(* CODESYS project MC508.project
   Title: MC508
   CompiledLibraryCompatibilityVersion: LeadSysStudio V3.5 SP15 Patch 4

Project tree, tasks and I/O mapping:
  Device : MC508, Leadshine Technology Co., Ltd., order no. 508101, version 3.5.15.40
      settings: RetainMode = 0; RetainStartAddr = 20480; RetainEndAddr = 524288; RetainSize = 524288
    application Application
      libraries: Standard, * (System); VisuDialogs, * (System); LS_ModbusMasterlib, 0.0.0.2 (Leadshine Technology Co.Ltd)
      task MainTask (cyclic, interval 500 µs, priority 1) calls main
      program main [ST]: io, vfd_setup, motion, save_apply, vfd, save_check, cut, supply, extract, work, stick
      visualisation Visualization
      Symbols
      function StateNext [ST]
      Object/
        data type Cylinder
        data type Button
      Enum/
        data type State
        data type VFDType
      DataMain/
        data type HMIData
        data type SaveData
        data type VFDData
      DataWork/
        data type CutData
        data type SupplyData
        data type ExtractData
        data type WorkData
        data type StickData
    Device Diagnose
    Network Configuration
      LocalBus Config
    Resource Usage
    SoftMotion General Axis Pool
      LS_Axis_0 : Axis, 3S - Smart Software Solutions GmbH, order no. 1805, version 4.0.0.0
          settings: eRampType = 3; fSWLimitPositive = 0.0
      LS_Axis_1 : Axis, 3S - Smart Software Solutions GmbH, order no. 1805, version 4.0.0.0
          settings: wDriveID = 2; eRampType = 3
    High_Speed_IO_Module : High Speed IO, Leadshine Technology Co., Ltd., version 3.5.15.40
        settings: HS_IO_Mode_0.High Out IO Mode 0 = 65537; HS_IO_Mode_0.High Out IO Mode 1 = 65537; Axis_Mask = 3; Ioout_Mask = 15; Axis_0_Pulse_FPGA_Config.Axis Ratio Nume = 1000; Axis_0_Pulse_FPGA_Config.Axis Ratio Denom = 1000; Axis_1_Pulse_FPGA_Config.Axis Ratio Nume = 1000; Axis_1_Pulse_FPGA_Config.Axis Ratio Denom = 50000
        unmapped channels: Genral_IO_IN, Genral_IO_Out
    LocalBus_Master_Module : LocalBus Master, Leadshine Technology Co., Ltd., version 3.5.15.40
  text list GlobalTextList
*)

// Device/Application/DataMain/HMIData
TYPE HMIData :
STRUCT
	plc_ready: BOOL;
	hmi_ready: BOOL;
	run: BOOL;
	stop: BOOL;
	//
	supply_run_press: BOOL;
	supply_run_glue: BOOL;
	supply_run_conveyer: BOOL;
	supply_run_roll: BOOL;
	stick_run_press: BOOL;
	stick_run_roll: BOOL;
	cut_run: BOOL;
	extract_run: BOOL;
	//
	supply_press_a: BOOL;
	supply_press_b: BOOL;
	stick_press: BOOL;
	cut_press: BOOL;
	//
	vfds_run: ARRAY[0..15] OF BOOL;
	//
	save_data: SaveData;
	save: BOOL;
	save_need_check: BOOL;
	save_need: BOOL;
	//
	view_stop: BOOL;
	view_halt: BOOL;
	view_can_run: BOOL;
	view_can_stop: BOOL;
	view_supply_roll_is_long: BOOL;
	view_supply_roll_is_short: BOOL;
	view_supply_select_roll: BOOL;
	view_stick_foil_in: BOOL;
	view_stick_roll_speed_micron_per_sec: UDINT;
	view_cut_foil_in: BOOL;
	view_cut_position: DINT;
	view_cut_speed_micron_per_sec: UDINT;
	view_cut_servo_is_ready: BOOL;
	view_cut_servo_is_home: BOOL;
	view_extract_foil_in: BOOL;
	view_extract_reach: BOOL;
	//
	view_state_main: INT;
	view_state_work: INT;
	//
	view_state_supply_press: INT;
	view_state_supply_glue: INT;
	view_state_supply_conveyer: INT;
	view_state_supply_roll: INT;
	view_state_stick_press: INT;
	view_state_stick_roll: INT;
	view_state_cut: INT;
	view_state_extract: INT;
	//
	view_vfds_f_target: ARRAY[0..15] OF UINT;
END_STRUCT
END_TYPE

// Device/Application/Enum/State
{attribute 'qualified_only'}
{attribute 'strict'}
TYPE State : (
	NONE := 0,
	RST := 1,
	RST_DONE := 50,
	HOME := 51,
	HOME_FORWARD := 71,
	HOME_DONE := 99,
	READY := 100,
	RUN := 101,
	RUN_ING := 200
);
END_TYPE

// Device/Application/DataMain/SaveData
TYPE SaveData :
STRUCT
	set_done: BOOL;
	main_frequency: UINT;
	stick_speed_factor: UDINT;
	stick_roll_gear_ratio: UDINT;
	stick_roll_diameter_micron: UDINT;
	stick_stop_distance_micron: UDINT; // distance after panel's tail move out of sensor
	cut_angle_radian: UDINT;
	cut_length_micron: UDINT;
	cut_accel_decel_time: UINT;
	cut_run_distance_micron: UINT; // distance after panel's head enter sensor
	vfds_frequency_factor: ARRAY[0..15] OF UINT;
END_STRUCT
END_TYPE

// Device/Application/DataWork/CutData
TYPE CutData :
STRUCT
	state: INT;
	press: Cylinder;
	servo_on: BOOL;
	servo_is_ready: BOOL;
	servo_is_home: BOOL;
	foil_in_rise: R_TRIG;
	foil_in_fall: F_TRIG;
	blade_vfd_id: USINT;
	speed_target: LREAL; // micron per sec
	speed_factor: LREAL; // speed_factor = current_velocity / target_velocity
	speed_factor_active: BOOL;
	travel_length_micron: LREAL; // travel_length = cut_length / cos(angle_radian)
	accel_decel_time: LREAL;
	angle_radian: LREAL;
	run: Button;
	//
	sin_cut_angle: LREAL;
	home_zero_position: LREAL;
	stick_axis_target_position: LREAL;
END_STRUCT
END_TYPE

// Device/Application/DataMain/VFDData
TYPE VFDData :
STRUCT
	vfds_type: ARRAY[0..15] OF INT;
	i: USINT;
	i_control: UINT;
	i_frequency: DINT;
END_STRUCT
END_TYPE

// Device/Application/DataWork/SupplyData
TYPE SupplyData :
STRUCT
	state_press: INT;
	press_a: Cylinder;
	press_b: Cylinder;
	run_press: Button;
	//
	state_glue: INT;
	glues_vfd_id: ARRAY[0..1] OF USINT;
	run_glue: Button;
	//
	state_conveyer: INT;
	conveyers_vfd_id: ARRAY[0..1] OF USINT;
	run_conveyer: Button;
	//
	state_roll: INT;
	rolls_vfd_id: ARRAY[0..1] OF USINT;
	roll_index: USINT;
	roll_is_long: BOOL;
	roll_is_short: BOOL;
	roll_is_short_timer: TON;
	select_roll: BOOL;
	run_roll: Button;
END_STRUCT
END_TYPE

// Device/Application/DataWork/ExtractData
TYPE ExtractData :
STRUCT
	state: INT;
	foil_in_rise: R_TRIG;
	reach_rise: R_TRIG;
	conveyers_vfd_id: ARRAY[0..1] OF USINT;
	blades_vfd_id: ARRAY[0..1] OF USINT;
	run: Button;
END_STRUCT
END_TYPE

// Device/Application/DataWork/WorkData
TYPE WorkData :
STRUCT
	state: INT;
	run: Button;
	can_run: BOOL;
	stop: Button;
	can_stop: BOOL;
	halt: Button;
END_STRUCT
END_TYPE

// Device/Application/DataWork/StickData
TYPE StickData :
STRUCT
	state_press: INT;
	state_roll: INT;
	press: Cylinder;
	foil_in_rise: R_TRIG;
	foil_in_fall: F_TRIG;
	run_press: Button;
	run_roll: Button;
	speed_target: LREAL; // 1000 ppr -> 3000 rpm = 50_000
	speed_micron_per_sec: LREAL;
	//
	micron_per_servo_round: LREAL;
	stop_distance: LREAL;
END_STRUCT
END_TYPE

// Device/Application/Object/Cylinder
TYPE Cylinder :
STRUCT
	on: BOOL;
	n_timer: TON;
	p_timer: TON;
END_STRUCT
END_TYPE

// Device/Application/Object/Button
TYPE Button :
STRUCT
	rise: R_TRIG;
	fall: F_TRIG;
END_STRUCT
END_TYPE

// Device/Application/Enum/VFDType
{attribute 'qualified_only'}
{attribute 'strict'}
TYPE VFDType :
(
	NORMAL := 0,
	SPINDLE := 1,
	CUSTOM := 2
);
END_TYPE

// Device/Application/main
PROGRAM main
VAR
	axis_stick: POINTER TO SM3_Basic.AXIS_REF_VIRTUAL_SM3;
	axis_stick_power: MC_Power;
	axis_stick_stop: MC_Stop;
	axis_stick_reset: MC_Reset;
	axis_stick_set_position: MC_SetPosition;
	axis_stick_mv: MC_MoveVelocity;
	axis_stick_fv: SMC_FollowVelocity;
	//
	axis_cut: POINTER TO SM3_Basic.AXIS_REF_VIRTUAL_SM3;
	axis_cut_power: MC_Power;
	axis_cut_stop: MC_Stop;
	axis_cut_reset: MC_Reset;
	axis_cut_set_position: MC_SetPosition;
	axis_cut_mabs: MC_MoveAbsolute;
	//
	state_main: INT;
	main_save: Button;
	supply_data: SupplyData;
	stick_data: StickData;
	cut_data: CutData;
	extract_data: ExtractData;
	work_data: WorkData;
	hmi_data: HMIData;
	//
	vfd_master: LS_ModbusMaster;
	vfd_para: SerialCommunicationPara;
	vfd_configs: ARRAY [0..127] OF ModbusConfig;
	vfd_data: VFDData;
END_VAR

VAR CONSTANT
	c_vfd_count: BYTE := 11;
	c_main_frequency_min: UINT := 10_00;
	c_main_frequency_max: UINT := 50_00;
	c_axis_stick_max_speed: LREAL := 3000.0 * 1000.0 / 60.0; // 3000rpm, 1000 ppr at servo
	c_axis_cut_max_speed: LREAL := 4920.0 * 50_000.0 / 60.0; // 4920rpm, 1000 ppr at servo
	c_axis_cut_home_speed_micron_per_sec: LREAL := 20_000.0;
	c_axis_cut_home_offset_micron: LREAL := 10_000.0;
	c_axis_stick_ramp_time_sec: LREAL := 0.1;
	c_dt: LREAL := 0.000_500;
END_VAR

VAR RETAIN
	save_data: SaveData;
END_VAR

CASE state_main OF
	State.NONE:
		axis_stick := ADR(LS_Axis_0);
		axis_cut := ADR(LS_Axis_1);
		supply_data.press_a.on := TRUE;
		axis_stick_fv.fSetVelocity := 0.0;
		vfd_setup();
		StateNext(state_main);
	1:
		axis_stick_power.Enable := TRUE;
		axis_stick_power.bDriveStart := TRUE;
		axis_stick_power.bRegulatorOn := TRUE;
		axis_cut_power.Enable := TRUE;
		axis_cut_power.bDriveStart := TRUE;
		axis_cut_power.bRegulatorOn := TRUE;
		StateNext(state_main);
	2:
		IF NOT save_data.set_done THEN
			save_data.set_done := TRUE;
			save_data.main_frequency := 50_00;
			save_data.stick_speed_factor := 1_000;
			save_data.stick_roll_gear_ratio := 20_000;
			save_data.stick_roll_diameter_micron := 120_000;
			save_data.stick_stop_distance_micron := 0_001;
			save_data.cut_angle_radian := 0_230_500;
			save_data.cut_length_micron := 290_000;
			save_data.cut_accel_decel_time := 0_100;
			save_data.cut_run_distance_micron := 20_000;
			//
			save_data.vfds_frequency_factor[supply_data.glues_vfd_id[0]] := 1_000;
			save_data.vfds_frequency_factor[supply_data.glues_vfd_id[1]] := 1_000;
			save_data.vfds_frequency_factor[supply_data.conveyers_vfd_id[0]] := 1_000;
			save_data.vfds_frequency_factor[supply_data.conveyers_vfd_id[1]] := 1_000;
			save_data.vfds_frequency_factor[supply_data.rolls_vfd_id[0]] := 0_500;
			save_data.vfds_frequency_factor[supply_data.rolls_vfd_id[1]] := 0_500;
			save_data.vfds_frequency_factor[cut_data.blade_vfd_id] := 50_00;
			save_data.vfds_frequency_factor[extract_data.conveyers_vfd_id[0]] := 50_00;
			save_data.vfds_frequency_factor[extract_data.conveyers_vfd_id[1]] := 50_00;
			save_data.vfds_frequency_factor[extract_data.blades_vfd_id[0]] := 200_00;
			save_data.vfds_frequency_factor[extract_data.blades_vfd_id[1]] := 200_00;
		END_IF
		StateNext(state_main);
	3:
		save_apply();
		StateNext(state_main);
	4:
		hmi_data.plc_ready := TRUE;
		work_data.state := State.RST;
		state_main := State.RUN_ING;
	State.RUN_ING:
		motion();
		io();
		vfd();
		work();
		supply();
		stick();
		cut();
		extract();
END_CASE

ACTION io:
work_data.can_run := work_data.stop.fall.CLK AND work_data.halt.rise.CLK AND work_data.state = State.READY;
work_data.can_stop := work_data.state >= State.RUN;
////////////
//HMI DOWN//
///////////
IF hmi_data.hmi_ready THEN
	////////
	//WORK//
	////////
	work_data.run.rise(CLK:= hmi_data.run, Q=> );
	IF work_data.run.rise.Q AND work_data.can_run THEN
		work_data.state := State.RUN;
	END_IF
	work_data.stop.rise(CLK:= hmi_data.stop, Q=> );
	IF work_data.stop.rise.Q AND work_data.can_stop THEN
		work_data.state := State.RST;
	END_IF
	//////////
	//SUPPLY//
	//////////
	supply_data.run_press.rise(CLK:= hmi_data.supply_run_press, Q=> );
	IF supply_data.run_press.rise.Q THEN
		CASE supply_data.state_press OF
			State.NONE:
				supply_data.state_press := State.RST;
			State.READY:
				supply_data.state_press := State.RUN;
			State.RUN_ING:
				supply_data.state_press := State.RST;
		END_CASE
	END_IF
	supply_data.run_glue.rise(CLK:= hmi_data.supply_run_glue, Q=> );
	IF supply_data.run_glue.rise.Q THEN
		CASE supply_data.state_glue OF
			State.NONE:
				supply_data.state_glue := State.RST;
			State.READY:
				supply_data.state_glue := State.RUN;
			State.RUN_ING:
				supply_data.state_glue := State.RST;
		END_CASE
	END_IF
	supply_data.run_conveyer.rise(CLK:= hmi_data.supply_run_conveyer, Q=> );
	IF supply_data.run_conveyer.rise.Q THEN
		CASE supply_data.state_conveyer OF
			State.NONE:
				supply_data.state_conveyer := State.RST;
			State.READY:
				supply_data.state_conveyer := State.RUN;
			State.RUN_ING:
				supply_data.state_conveyer := State.RST;
		END_CASE
	END_IF
	supply_data.run_roll.rise(CLK:= hmi_data.supply_run_roll, Q=> );
	IF supply_data.run_roll.rise.Q THEN
		CASE supply_data.state_roll OF
			State.NONE:
				supply_data.state_roll := State.RST;
			State.READY:
				supply_data.state_roll := State.RUN;
			State.RUN_ING:
				supply_data.state_roll := State.RST;
		END_CASE
	END_IF
	/////////
	//STICK//
	/////////
	stick_data.run_press.rise(CLK:= hmi_data.stick_run_press, Q=> );
	IF stick_data.run_press.rise.Q THEN
		CASE stick_data.state_press OF
			State.NONE:
				stick_data.state_press := State.RST;
			State.READY:
				stick_data.state_press := State.RUN;
			State.RUN_ING:
				stick_data.state_press := State.RST;
		END_CASE
	END_IF
	stick_data.run_roll.rise(CLK:= hmi_data.stick_run_roll, Q=> );
	IF stick_data.run_roll.rise.Q THEN
		CASE stick_data.state_roll OF
			State.NONE:
				stick_data.state_roll := State.RST;
			State.RST_DONE:
				stick_data.state_roll := State.HOME;
			State.HOME_DONE:
				stick_data.state_roll := State.READY;
			State.READY:
				stick_data.state_roll := State.RST;
		END_CASE
	END_IF
	///////
	//CUT//
	///////
	cut_data.run.rise(CLK:= hmi_data.cut_run, Q=> );
	IF cut_data.run.rise.Q THEN
		CASE cut_data.state OF
			State.NONE:
				cut_data.state := State.RST;
			State.RST_DONE:
				cut_data.state := State.HOME;
			State.HOME_DONE:
				cut_data.state := State.READY;
			State.READY:
				cut_data.state := State.RST;
		END_CASE
	END_IF
	///////////
	//EXTRACT//
	///////////
	extract_data.run.rise(CLK:= hmi_data.extract_run, Q=> );
	IF extract_data.run.rise.Q THEN
		CASE extract_data.state OF
			State.NONE:
				extract_data.state := State.RST;
			State.RST_DONE:
				extract_data.state := State.HOME;
			State.HOME_DONE:
				extract_data.state := State.READY;
			State.READY:
				extract_data.state := State.RST;
		END_CASE
	END_IF
	////////
	//SAVE//
	////////
	IF hmi_data.save_need_check THEN
		save_check();
		hmi_data.save_need_check := FALSE;
	END_IF
	main_save.rise(CLK:= hmi_data.save, Q=> );
	IF main_save.rise.Q THEN
		save_data := hmi_data.save_data;
		save_apply();
		hmi_data.save_need := FALSE;
		hmi_data.save := FALSE;
	END_IF
END_IF
/////////
//INPUT//
/////////
supply_data.roll_is_long := %IX0.4;
supply_data.roll_is_short := %IX0.5;
work_data.halt.rise(CLK:= %IX1.4, Q=> );
supply_data.select_roll := %IX1.5;
//
stick_data.foil_in_rise(CLK:= NOT %IX0.6, Q=> );
stick_data.foil_in_fall(CLK:= stick_data.foil_in_rise.CLK, Q=> );
//
cut_data.servo_is_ready := %IX0.1;
cut_data.servo_is_home := NOT %IX0.7;
cut_data.foil_in_rise(CLK:= %IX1.0, Q=> );
cut_data.foil_in_fall(CLK:= cut_data.foil_in_rise.CLK, Q=> );
//
extract_data.foil_in_rise(CLK:= %IX1.1, Q=> );
extract_data.reach_rise(CLK:= %IX1.2, Q=> );
//
work_data.stop.fall(CLK:= %IX1.7, Q=> );
IF work_data.stop.fall.Q AND work_data.can_stop THEN
	work_data.state := State.RST;
END_IF
//
supply_data.press_a.n_timer(IN:= NOT supply_data.press_a.on, PT:= , Q=> , ET=> );
supply_data.press_a.p_timer(IN:= supply_data.press_a.on, PT:= , Q=> , ET=> );
supply_data.press_b.n_timer(IN:= NOT supply_data.press_b.on, PT:= , Q=> , ET=> );
supply_data.press_b.p_timer(IN:= supply_data.press_b.on, PT:= , Q=> , ET=> );
supply_data.roll_is_short_timer(IN:= supply_data.roll_is_short, PT:= , Q=> , ET=> );
stick_data.press.n_timer(IN:= NOT stick_data.press.on, PT:= , Q=> , ET=> );
stick_data.press.p_timer(IN:= stick_data.press.on, PT:= , Q=> , ET=> );
cut_data.press.n_timer(IN:= NOT cut_data.press.on, PT:= , Q=> , ET=> );
cut_data.press.p_timer(IN:= cut_data.press.on, PT:= , Q=> , ET=> );
//////////
//OUTPUT//
//////////
%QX1.4 := NOT supply_data.press_a.on;
%QX1.5 := supply_data.press_b.on;
%QX1.6 := stick_data.press.on;
%QX1.2 := cut_data.servo_on;
%QX1.7 := NOT cut_data.press.on;
//////////
//HMI UP//
//////////
IF hmi_data.hmi_ready THEN
	hmi_data.view_stop := work_data.stop.fall.CLK;
	hmi_data.view_halt := work_data.halt.rise.CLK;
	hmi_data.view_can_run := work_data.can_run;
	hmi_data.view_can_stop := work_data.can_stop;
	hmi_data.view_supply_roll_is_long := supply_data.roll_is_long;
	hmi_data.view_supply_roll_is_short := supply_data.roll_is_short;
	hmi_data.view_supply_select_roll := supply_data.select_roll;
	hmi_data.view_stick_foil_in := NOT stick_data.foil_in_rise.CLK;
	hmi_data.view_stick_roll_speed_micron_per_sec := LREAL_TO_UDINT(stick_data.speed_micron_per_sec);
	hmi_data.view_cut_foil_in := cut_data.foil_in_fall.CLK;
	hmi_data.view_cut_position := LREAL_TO_DINT(axis_cut^.fActPosition);
	hmi_data.view_cut_speed_micron_per_sec := LREAL_TO_UDINT(cut_data.speed_target);
	hmi_data.view_cut_servo_is_ready := cut_data.servo_is_ready;
	hmi_data.view_cut_servo_is_home := NOT cut_data.servo_is_home;
	hmi_data.view_extract_foil_in := extract_data.foil_in_rise.CLK;
	hmi_data.view_extract_reach := extract_data.reach_rise.CLK;
	//
	hmi_data.view_state_main := state_main;
	hmi_data.view_state_work := work_data.state;
	//
	hmi_data.view_state_supply_press := supply_data.state_press;
	hmi_data.view_state_supply_glue := supply_data.state_glue;
	hmi_data.view_state_supply_conveyer := supply_data.state_conveyer;
	hmi_data.view_state_supply_roll := supply_data.state_roll;
	hmi_data.view_state_stick_press := stick_data.state_press;
	hmi_data.view_state_stick_roll := stick_data.state_roll;
	hmi_data.view_state_cut := cut_data.state;
	hmi_data.view_state_extract := extract_data.state;
	//
	FOR vfd_data.i := 0 TO (c_vfd_count - 1) BY 1 DO
		hmi_data.view_vfds_f_target[vfd_data.i] := vfd_configs[vfd_data.i].arwWriteData[1];
	END_FOR
	//
	IF work_data.state = State.READY THEN
		supply_data.press_a.on := hmi_data.supply_press_a;
		supply_data.press_b.on := hmi_data.supply_press_b;
		stick_data.press.on := hmi_data.stick_press;
		cut_data.press.on := hmi_data.cut_press;
	ELSE
		hmi_data.supply_press_a := supply_data.press_a.on;
		hmi_data.supply_press_b := supply_data.press_b.on;
		hmi_data.stick_press := stick_data.press.on;
		hmi_data.cut_press := cut_data.press.on;
	END_IF
END_IF
END_ACTION

ACTION vfd_setup:
vfd_para.udiPort := 3; // 2: COM2: RS232, 3: COM0: RS485, 4: COM1: RS485
vfd_para.udiBaudrate := 57600;
vfd_para.udiByteSize := 8;
vfd_para.udiPARITY := LS_ModbusMasterlib.COM.PARITY.EVEN;
vfd_para.udiStopBits := LS_ModbusMasterlib.COM.STOPBIT.ONESTOPBIT;
vfd_para.udiTimeout := 1000;
//
vfd_master.byModbusConfigNumber := c_vfd_count;
//
FOR vfd_data.i := 0 TO 127 DO
	vfd_configs[vfd_data.i].xCycle := vfd_data.i < vfd_master.byModbusConfigNumber;
	vfd_configs[vfd_data.i].xTrigger := FALSE;
	vfd_configs[vfd_data.i].uiCycleTime := 10;
END_FOR
//
supply_data.glues_vfd_id[0] := 1; vfd_data.vfds_type[supply_data.glues_vfd_id[0]] := VFDType.NORMAL;
supply_data.glues_vfd_id[1] := 2; vfd_data.vfds_type[supply_data.glues_vfd_id[1]] := VFDType.NORMAL;
supply_data.conveyers_vfd_id[0] := 0; vfd_data.vfds_type[supply_data.conveyers_vfd_id[0]] := VFDType.NORMAL;
supply_data.conveyers_vfd_id[1] := 5; vfd_data.vfds_type[supply_data.conveyers_vfd_id[1]] := VFDType.NORMAL;
supply_data.rolls_vfd_id[0] := 3; vfd_data.vfds_type[supply_data.rolls_vfd_id[0]] := VFDType.NORMAL;
supply_data.rolls_vfd_id[1] := 4; vfd_data.vfds_type[supply_data.rolls_vfd_id[1]] := VFDType.NORMAL;
//
cut_data.blade_vfd_id := 6; vfd_data.vfds_type[cut_data.blade_vfd_id] := VFDType.SPINDLE;
//
extract_data.conveyers_vfd_id[0] := 7; vfd_data.vfds_type[extract_data.conveyers_vfd_id[0]] := VFDType.CUSTOM;
extract_data.conveyers_vfd_id[1] := 8; vfd_data.vfds_type[extract_data.conveyers_vfd_id[1]] := VFDType.CUSTOM;
extract_data.blades_vfd_id[0] := 9; vfd_data.vfds_type[extract_data.blades_vfd_id[0]] := VFDType.SPINDLE;
extract_data.blades_vfd_id[1] := 10; vfd_data.vfds_type[extract_data.blades_vfd_id[1]] := VFDType.SPINDLE;
//
FOR vfd_data.i := 0 TO (c_vfd_count - 1) BY 1 DO
	vfd_data.i := vfd_data.i;
	hmi_data.vfds_run[vfd_data.i] := FALSE;
END_FOR
END_ACTION

ACTION motion:
LS_MotionControl_P(stAxis=> ,xClearErr=> ,fLimtAxisSpeedJump=> ,xDone=> ,xError=> ,eErrorID=> ,xLimitAxisMoveFlag=> );
//
LS_MotionControl_P.stAxis.PulAxis_0 := axis_stick;
axis_stick_power(Axis:= axis_stick^, Enable:= , bRegulatorOn:= , bDriveStart:= , Status=> , bRegulatorRealState=> , bDriveStartRealState=> , Busy=> , Error=> , ErrorID=> );
axis_stick_stop(Axis:= axis_stick^, Execute:= , Deceleration:= , Jerk:= , Done=> , Busy=> , Error=> , ErrorID=> );
axis_stick_reset(Axis:= axis_stick^, Execute:= , Done=> , Busy=> , Error=> , ErrorID=> );
axis_stick_set_position(Axis:= axis_stick^, Execute:= , Position:= , Mode:= , Done=> , Busy=> , Error=> , ErrorID=> );
axis_stick_mv(Axis:= axis_stick^, Execute:= , Velocity:= , Acceleration:= , Deceleration:= , Jerk:= , Direction:= , BufferMode:= , InVelocity=> , Busy=> , Active=> , CommandAborted=> , Error=> , ErrorID=> );
axis_stick_fv(Axis:= axis_stick^, bExecute:= , fSetVelocity:= , bBusy=> , bCommandAborted=> , bError=> , iErrorID=> );
//
LS_MotionControl_P.stAxis.PulAxis_1 := axis_cut;
axis_cut_power(Axis:= axis_cut^, Enable:= , bRegulatorOn:= , bDriveStart:= , Status=> , bRegulatorRealState=> , bDriveStartRealState=> , Busy=> , Error=> , ErrorID=> );
axis_cut_stop(Axis:= axis_cut^, Execute:= , Deceleration:= , Jerk:= , Done=> , Busy=> , Error=> , ErrorID=> );
axis_cut_reset(Axis:= axis_cut^, Execute:= , Done=> , Busy=> , Error=> , ErrorID=> );
axis_cut_set_position(Axis:= axis_cut^, Execute:= , Position:= , Mode:= , Done=> , Busy=> , Error=> , ErrorID=> );
axis_cut_mabs(Axis:= axis_cut^, Execute:= , Position:= , Velocity:= , Acceleration:= , Deceleration:= , Jerk:= , Direction:= , BufferMode:= , Done=> , Busy=> , Active=> , CommandAborted=> , Error=> , ErrorID=> );
END_ACTION

ACTION save_apply:
save_data.main_frequency := MAX(c_main_frequency_min, MIN(c_main_frequency_max, save_data.main_frequency));
save_data.stick_speed_factor := MAX(0_100, MIN(1_000, save_data.stick_speed_factor));
save_data.stick_roll_gear_ratio := MAX(1_000, MIN(30_000, save_data.stick_roll_gear_ratio));
save_data.stick_roll_diameter_micron := MAX(100_000, MIN(140_000, save_data.stick_roll_diameter_micron));
save_data.stick_stop_distance_micron := MAX(0_001, MIN(50_000, save_data.stick_stop_distance_micron));
save_data.cut_angle_radian := MAX(0_100_000, MIN(1_000_000, save_data.cut_angle_radian));
save_data.cut_length_micron := MAX(200_000, MIN(300_000, save_data.cut_length_micron));
save_data.cut_accel_decel_time := MAX(0_100, MIN(0_500, save_data.cut_accel_decel_time));
save_data.cut_run_distance_micron := MAX(1_000, MIN(50_000, save_data.cut_run_distance_micron));
//
stick_data.speed_target := UDINT_TO_LREAL(save_data.stick_speed_factor * save_data.main_frequency) * 1E-2;
IF stick_data.speed_target > c_axis_stick_max_speed THEN
	stick_data.speed_target := c_axis_stick_max_speed;
END_IF
stick_data.micron_per_servo_round := (save_data.stick_roll_diameter_micron * PI) / (UDINT_TO_LREAL(save_data.stick_roll_gear_ratio) * 1E-3);
stick_data.speed_micron_per_sec := stick_data.micron_per_servo_round * stick_data.speed_target * 1E-3;
cut_data.angle_radian := UDINT_TO_LREAL(save_data.cut_angle_radian) * 1E-6;
cut_data.sin_cut_angle := SIN(cut_data.angle_radian);
cut_data.speed_target := stick_data.speed_micron_per_sec / cut_data.sin_cut_angle;
IF cut_data.speed_target > c_axis_cut_max_speed THEN
	cut_data.speed_target := c_axis_cut_max_speed;
	stick_data.speed_micron_per_sec := cut_data.speed_target * cut_data.sin_cut_angle;
	save_data.stick_speed_factor := LREAL_TO_UINT(
		stick_data.speed_micron_per_sec * 1E3 / stick_data.micron_per_servo_round
		* 1E2 / save_data.main_frequency
	);
	save_data.stick_speed_factor := MAX(0_100, MIN(1_000, save_data.stick_speed_factor));
END_IF
cut_data.accel_decel_time := UINT_TO_LREAL(save_data.cut_accel_decel_time) * 1E-3;
cut_data.travel_length_micron := UDINT_TO_LREAL(save_data.cut_length_micron) / COS(cut_data.angle_radian);
//
supply_data.press_a.n_timer.PT := INT_TO_TIME(0_800);
supply_data.press_a.p_timer.PT := INT_TO_TIME(0_800);
supply_data.press_b.n_timer.PT := INT_TO_TIME(0_800);
supply_data.press_b.p_timer.PT := INT_TO_TIME(0_800);
supply_data.roll_is_short_timer.PT := INT_TO_TIME(2_000);
stick_data.press.n_timer.PT := INT_TO_TIME(0_800);
stick_data.press.p_timer.PT := INT_TO_TIME(0_800);
cut_data.press.n_timer.PT := INT_TO_TIME(0_100);
cut_data.press.p_timer.PT := INT_TO_TIME(0_100);
//
FOR vfd_data.i := 0 TO (c_vfd_count - 1) BY 1 DO
	CASE vfd_data.vfds_type[vfd_data.i] OF
		VFDType.NORMAL:
			vfd_data.i_frequency := MAX(0_100, MIN(1_000, save_data.vfds_frequency_factor[vfd_data.i]));
		VFDType.SPINDLE:
			vfd_data.i_frequency := MAX(50_00, MIN(200_00, save_data.vfds_frequency_factor[vfd_data.i]));
		VFDType.CUSTOM:
			vfd_data.i_frequency := MAX(c_main_frequency_min, MIN(80_00, save_data.vfds_frequency_factor[vfd_data.i]));
	END_CASE
	save_data.vfds_frequency_factor[vfd_data.i] := DINT_TO_UINT(vfd_data.i_frequency);
END_FOR
//FINAL
hmi_data.save_data := save_data;
END_ACTION

ACTION vfd:
vfd_master(
	arstModbusConfig:= vfd_configs, 
	stSerialCommunicationPara:= vfd_para, 
	byModbusConfigNumber=> , 
	xError=> , 
	ErrorID=> );
FOR vfd_data.i := 0 TO (c_vfd_count - 1) BY 1 DO
	CASE vfd_data.vfds_type[vfd_data.i] OF
		VFDType.NORMAL:
			vfd_data.i_frequency := (save_data.vfds_frequency_factor[vfd_data.i] * save_data.main_frequency) / 1_000;
		VFDType.SPINDLE:
			vfd_data.i_frequency := save_data.vfds_frequency_factor[vfd_data.i];
		VFDType.CUSTOM:
			vfd_data.i_frequency := save_data.vfds_frequency_factor[vfd_data.i];
	END_CASE
	IF hmi_data.vfds_run[vfd_data.i] THEN
		vfd_data.i_control := 1;
	ELSE
		vfd_data.i_control := 5;
	END_IF
	vfd_configs[vfd_data.i].usiAddress := vfd_data.i + 1;
	vfd_configs[vfd_data.i].usiFunctionCode := ModbusFuntionCode.Write_Muluiple_Register;
	vfd_configs[vfd_data.i].wOffset := 16#2000;
	vfd_configs[vfd_data.i].wLength := 2;
	vfd_configs[vfd_data.i].arwWriteData[0] := vfd_data.i_control;
	vfd_configs[vfd_data.i].arwWriteData[1] := DINT_TO_UINT(vfd_data.i_frequency);
END_FOR
END_ACTION

ACTION save_check:
hmi_data.save_need := (
	save_data.main_frequency <> hmi_data.save_data.main_frequency OR
	save_data.stick_speed_factor <> hmi_data.save_data.stick_speed_factor OR
	save_data.stick_roll_gear_ratio <> hmi_data.save_data.stick_roll_gear_ratio OR
	save_data.stick_roll_diameter_micron <> hmi_data.save_data.stick_roll_diameter_micron OR
	save_data.stick_stop_distance_micron <> hmi_data.save_data.stick_stop_distance_micron OR
	save_data.cut_angle_radian <> hmi_data.save_data.cut_angle_radian OR
	save_data.cut_length_micron <> hmi_data.save_data.cut_length_micron OR
	save_data.cut_accel_decel_time <> hmi_data.save_data.cut_accel_decel_time OR
	save_data.cut_run_distance_micron <> hmi_data.save_data.cut_run_distance_micron
);
FOR vfd_data.i := 0 TO (c_vfd_count - 1) BY 1 DO
	IF save_data.vfds_frequency_factor[vfd_data.i] <> hmi_data.save_data.vfds_frequency_factor[vfd_data.i] THEN
		hmi_data.save_need := TRUE;
	END_IF
END_FOR
END_ACTION

ACTION cut:
cut_data.speed_factor_active := FALSE;
//
CASE cut_data.state OF
	State.RST:
		hmi_data.vfds_run[cut_data.blade_vfd_id] := FALSE;
		IF axis_cut_mabs.Busy THEN
			axis_cut_stop.Deceleration := cut_data.speed_target / 0.1;
			axis_cut_stop.Jerk := axis_cut_stop.Deceleration * 5.0;
			axis_cut_stop.Execute := TRUE;
			StateNext(cut_data.state);
		ELSE
			cut_data.state := 3;
		END_IF
	2:
		IF axis_cut_stop.Done THEN
			axis_cut_stop.Execute := FALSE;
			axis_cut_mabs.Execute := FALSE;
			cut_data.state := 3;
		END_IF
	3:
		cut_data.press.on := FALSE;
		cut_data.servo_on := FALSE;
		StateNext(cut_data.state);
	4:
		IF cut_data.press.n_timer.Q THEN
			cut_data.state := State.RST_DONE;
		END_IF
	//////\\
	////\\\\
	//\\\\\\
	State.HOME:
		IF axis_cut_power.Status THEN
			cut_data.press.on := FALSE;
			cut_data.servo_on := TRUE;
			hmi_data.vfds_run[cut_data.blade_vfd_id] := TRUE;
			StateNext(cut_data.state);
		END_IF
	52:
		IF cut_data.press.n_timer.Q THEN
			StateNext(cut_data.state);
		END_IF
	53:
		IF cut_data.servo_is_home THEN
			cut_data.state := State.HOME_FORWARD;
		ELSE
			axis_cut_mabs.Position := axis_cut^.fActPosition - 1_000_000;
			axis_cut_mabs.Velocity := c_axis_cut_home_speed_micron_per_sec;
			axis_cut_mabs.Acceleration := axis_cut_mabs.Deceleration := axis_cut_mabs.Velocity / 0.1;
			axis_cut_mabs.Jerk := axis_cut_mabs.Acceleration * 5.0;
			//
			axis_cut_stop.Deceleration := axis_cut_mabs.Velocity / 0.1;
			axis_cut_stop.Jerk := axis_cut_stop.Deceleration * 5.0;
			//
			axis_cut_mabs.Execute := TRUE;
			StateNext(cut_data.state);
		END_IF
	54:
		IF cut_data.servo_is_home THEN
			axis_cut_stop.Execute := TRUE;
			StateNext(cut_data.state);
		END_IF
	55:
		IF axis_cut_stop.Done THEN
			axis_cut_stop.Execute := FALSE;
			axis_cut_mabs.Execute := FALSE;
			cut_data.state := State.HOME_FORWARD;
		END_IF
	State.HOME_FORWARD:
		axis_cut_mabs.Position := axis_cut^.fActPosition + 100_000;
		axis_cut_mabs.Velocity := c_axis_cut_home_speed_micron_per_sec * 0.25;
		axis_cut_mabs.Acceleration := axis_cut_mabs.Velocity / 0.1;
		axis_cut_mabs.Deceleration := axis_cut_mabs.Acceleration;
		axis_cut_mabs.Jerk := axis_cut_mabs.Acceleration * 5.0;
		//
		axis_cut_stop.Deceleration := axis_cut_mabs.Velocity / 0.1;
		axis_cut_stop.Jerk := axis_cut_stop.Deceleration * 5.0;
		//
		axis_cut_mabs.Execute := TRUE;
		StateNext(cut_data.state);
	72:
		IF NOT cut_data.servo_is_home THEN
			cut_data.home_zero_position := axis_cut^.fActPosition;
			axis_cut_stop.Execute := TRUE;
			StateNext(cut_data.state);
		END_IF
	73:
		IF axis_cut_stop.Done THEN
			axis_cut_stop.Execute := FALSE;
			axis_cut_mabs.Execute := FALSE;
			StateNext(cut_data.state);
		END_IF
	74:
		axis_cut_mabs.Position := cut_data.home_zero_position + c_axis_cut_home_offset_micron;
		axis_cut_mabs.Velocity := c_axis_cut_home_speed_micron_per_sec * 2;
		axis_cut_mabs.Acceleration := axis_cut_mabs.Velocity / 0.1;
		axis_cut_mabs.Deceleration := axis_cut_mabs.Acceleration;
		axis_cut_mabs.Jerk := axis_cut_mabs.Acceleration * 5.0;
		//
		axis_cut_stop.Deceleration := axis_cut_mabs.Velocity / 0.1;
		axis_cut_stop.Jerk := axis_cut_stop.Deceleration * 5.0;
		//
		axis_cut_mabs.Execute := TRUE;
		StateNext(cut_data.state);
	75:
		IF axis_cut_mabs.Done THEN
			axis_cut_mabs.Execute := FALSE;
			StateNext(cut_data.state);
		END_IF
	76:
		axis_cut_set_position.Position := 0.0;
		axis_cut_set_position.Execute := TRUE;
		StateNext(cut_data.state);
	77:
		IF axis_cut_set_position.Done THEN
			axis_cut_set_position.Execute := FALSE;
			cut_data.press.on := TRUE;
			StateNext(cut_data.state);
		END_IF
	78:
		IF cut_data.press.p_timer.Q THEN
			cut_data.state := State.HOME_DONE;
		END_IF
	//////\\
	////\\\\
	//\\\\\\
	State.READY:
		IF cut_data.foil_in_rise.Q THEN
			cut_data.stick_axis_target_position := (axis_stick^.fActPosition
				+ (UDINT_TO_LREAL(save_data.cut_run_distance_micron) / stick_data.micron_per_servo_round) * 1E3
			);
			cut_data.state := State.RUN;
		END_IF
	//////\\
	////\\\\
	//\\\\\\
	State.RUN:
		IF axis_stick^.fActPosition >= cut_data.stick_axis_target_position THEN
			axis_cut_mabs.Position := cut_data.travel_length_micron;
			axis_cut_mabs.Velocity := cut_data.speed_target;
			axis_cut_mabs.Acceleration := axis_cut_mabs.Velocity / cut_data.accel_decel_time;
			axis_cut_mabs.Deceleration := axis_cut_mabs.Acceleration;
			axis_cut_mabs.Jerk := axis_cut_mabs.Acceleration * 5.0;
			//
			axis_cut_stop.Deceleration := axis_cut_mabs.Velocity / cut_data.accel_decel_time;
			axis_cut_stop.Jerk := axis_cut_stop.Deceleration * 5.0;
			//
			axis_cut_mabs.Execute := TRUE;
			StateNext(cut_data.state);
		END_IF
	102:
		cut_data.speed_factor_active := TRUE;
		IF axis_cut_mabs.Done THEN
			axis_cut_mabs.Execute := FALSE;
			cut_data.press.on := FALSE;
			StateNext(cut_data.state);
		END_IF
	103:
		IF cut_data.press.n_timer.Q THEN
			StateNext(cut_data.state);
		END_IF
	104:
		axis_cut_mabs.Position := 0.0;
		axis_cut_mabs.Execute := TRUE;
		StateNext(cut_data.state);
	105:
		IF axis_cut_mabs.Done THEN
			axis_cut_mabs.Execute := FALSE;
			cut_data.press.on := TRUE;
			StateNext(cut_data.state);
		END_IF
	106:
		IF cut_data.press.p_timer.Q THEN
			cut_data.state := State.READY;
		END_IF
END_CASE
//
IF cut_data.speed_factor_active THEN
	cut_data.speed_factor := axis_cut^.fActVelocity / axis_cut_mabs.Velocity;
ELSE
	cut_data.speed_factor := 1.0;
END_IF
END_ACTION

ACTION supply:
/////////
//PRESS//
/////////
CASE supply_data.state_press OF
	//////\\
	////\\\\
	//\\\\\\
	State.RST:
		supply_data.press_b.on := FALSE;
		StateNext(supply_data.state_press);
	2:
		IF supply_data.press_b.n_timer.Q THEN
			supply_data.state_press := State.READY;
		END_IF
	//////\\
	////\\\\
	//\\\\\\
	State.RUN:
		supply_data.press_a.on := TRUE;
		StateNext(supply_data.state_press);
	102:
		IF supply_data.press_a.p_timer.Q THEN
			supply_data.press_b.on := TRUE;
			StateNext(supply_data.state_press);
		END_IF
	103:
		IF supply_data.press_b.p_timer.Q THEN
			supply_data.state_press := State.RUN_ING;
		END_IF
	//////\\
	////\\\\
	//\\\\\\
	State.RUN_ING:
		//
END_CASE

////////
//GLUE//
////////
CASE supply_data.state_glue OF
	State.RST:
		hmi_data.vfds_run[supply_data.glues_vfd_id[0]] := FALSE;
		hmi_data.vfds_run[supply_data.glues_vfd_id[1]] := FALSE;
		StateNext(supply_data.state_glue);
	2:
		supply_data.state_glue := State.READY;
	//////\\
	////\\\\
	//\\\\\\
	State.RUN:
		hmi_data.vfds_run[supply_data.glues_vfd_id[0]] := TRUE;
		hmi_data.vfds_run[supply_data.glues_vfd_id[1]] := TRUE;
		supply_data.state_glue := State.RUN_ING;
	//////\\
	////\\\\
	//\\\\\\
	State.RUN_ING:
		//
END_CASE

////////////
//CONVEYER//
////////////
CASE supply_data.state_conveyer OF
	State.RST:
		hmi_data.vfds_run[supply_data.conveyers_vfd_id[0]] := FALSE;
		hmi_data.vfds_run[supply_data.conveyers_vfd_id[1]] := FALSE;
		StateNext(supply_data.state_conveyer);
	2:
		supply_data.state_conveyer := State.READY;
	//////\\
	////\\\\
	//\\\\\\
	State.RUN:
		hmi_data.vfds_run[supply_data.conveyers_vfd_id[0]] := TRUE;
		hmi_data.vfds_run[supply_data.conveyers_vfd_id[1]] := TRUE;
		supply_data.state_conveyer := State.RUN_ING;
	//////\\
	////\\\\
	//\\\\\\
	State.RUN_ING:
		//
END_CASE

////////
//ROLL//
////////
CASE supply_data.state_roll OF
	State.RST:
		hmi_data.vfds_run[supply_data.rolls_vfd_id[0]] := FALSE;
		hmi_data.vfds_run[supply_data.rolls_vfd_id[1]] := FALSE;
		StateNext(supply_data.state_roll);
	2:
		supply_data.state_roll := State.READY;
	//////\\
	////\\\\
	//\\\\\\
	State.RUN:
		supply_data.roll_index := BOOL_TO_USINT(supply_data.select_roll);
		StateNext(supply_data.state_roll);
	102:
		supply_data.state_roll := State.RUN_ING;
	//////\\
	////\\\\
	//\\\\\\
	State.RUN_ING:
		IF supply_data.roll_is_short THEN
			hmi_data.vfds_run[supply_data.rolls_vfd_id[0]] := supply_data.roll_index = 0;
			hmi_data.vfds_run[supply_data.rolls_vfd_id[1]] := supply_data.roll_index = 1;
		END_IF
		IF supply_data.roll_is_long THEN
			hmi_data.vfds_run[supply_data.rolls_vfd_id[0]] := FALSE;
			hmi_data.vfds_run[supply_data.rolls_vfd_id[1]] := FALSE;
		END_IF
END_CASE
END_ACTION

ACTION extract:
CASE extract_data.state OF
	State.RST:
		hmi_data.vfds_run[extract_data.conveyers_vfd_id[0]] := FALSE;
		hmi_data.vfds_run[extract_data.conveyers_vfd_id[1]] := FALSE;
		hmi_data.vfds_run[extract_data.blades_vfd_id[0]] := FALSE;
		hmi_data.vfds_run[extract_data.blades_vfd_id[1]] := FALSE;
		StateNext(extract_data.state);
	2:
		extract_data.state := State.RST_DONE;
	//////\\
	////\\\\
	//\\\\\\
	State.HOME:
		hmi_data.vfds_run[extract_data.conveyers_vfd_id[0]] := TRUE;
		hmi_data.vfds_run[extract_data.conveyers_vfd_id[1]] := TRUE;
		hmi_data.vfds_run[extract_data.blades_vfd_id[0]] := TRUE;
		hmi_data.vfds_run[extract_data.blades_vfd_id[1]] := TRUE;
		StateNext(extract_data.state);
	52:
		IF extract_data.reach_rise.Q THEN
			hmi_data.vfds_run[extract_data.conveyers_vfd_id[1]] := FALSE;
			extract_data.state := State.HOME_DONE;
		END_IF
	//////\\
	////\\\\
	//\\\\\\
	State.READY:
		IF extract_data.foil_in_rise.Q THEN
			extract_data.state := State.RUN;
		END_IF
	//////\\
	////\\\\
	//\\\\\\
	State.RUN:
		hmi_data.vfds_run[extract_data.conveyers_vfd_id[1]] := TRUE;
		StateNext(extract_data.state);
	102:
		IF extract_data.reach_rise.Q THEN
			hmi_data.vfds_run[extract_data.conveyers_vfd_id[1]] := FALSE;
			StateNext(extract_data.state);
		END_IF
	103:
		extract_data.state := State.READY;
END_CASE
END_ACTION

ACTION work:
CASE work_data.state OF
	State.RST:
		supply_data.state_press := State.RST;
		supply_data.state_glue := State.RST;
		supply_data.state_conveyer := State.RST;
		supply_data.state_roll := State.RST;
		stick_data.state_press := State.RST;
		stick_data.state_roll := State.RST;
		cut_data.state := State.RST;
		extract_data.state := State.RST;
		StateNext(work_data.state);
	2:
		IF (	supply_data.state_press = State.READY AND
				supply_data.state_glue = State.READY AND
				supply_data.state_conveyer = State.READY AND
				supply_data.state_roll = State.READY AND
				stick_data.state_press = State.READY AND
				stick_data.state_roll = State.RST_DONE AND
				cut_data.state = State.RST_DONE AND
				extract_data.state = State.RST_DONE
			) THEN
			work_data.state := State.READY;
		END_IF
	//////\\
	////\\\\
	//\\\\\\
	State.READY:
		//check main.io for cylinder activation
	//////\\
	////\\\\
	//\\\\\\
	State.RUN:
		IF cut_data.servo_is_ready THEN
			StateNext(work_data.state);
		END_IF
	102:
		IF (	supply_data.state_press = State.READY AND
				stick_data.state_press = State.READY
			) THEN
			supply_data.state_press := State.RUN;
			stick_data.state_press := State.RUN;
			StateNext(work_data.state);
		END_IF 
	103:
		IF (
				supply_data.state_press = State.RUN_ING AND
				stick_data.state_press = State.RUN_ING
			) THEN
			stick_data.state_roll := State.HOME;
			cut_data.state := State.HOME;
			extract_data.state := State.HOME;
			StateNext(work_data.state);
		END_IF
	104:
		IF (	stick_data.state_roll = State.HOME_DONE AND
				cut_data.state = State.HOME_DONE AND
				extract_data.state = State.HOME_DONE
			) THEN
			stick_data.state_roll := State.READY;
			cut_data.state := State.READY;
			extract_data.state := State.READY;
			//
			supply_data.state_glue := State.RUN;
			supply_data.state_conveyer := State.RUN;
			supply_data.state_roll := State.RUN;
			StateNext(work_data.state);
		END_IF
	105:
		IF (	supply_data.state_glue = State.RUN_ING AND
				supply_data.state_conveyer = State.RUN_ING AND
				supply_data.state_roll = State.RUN_ING
			) THEN
			work_data.state := State.RUN_ING;
		END_IF
	//////\\
	////\\\\
	//\\\\\\
	State.RUN_ING:
		IF NOT work_data.halt.rise.CLK OR supply_data.roll_is_short_timer.Q THEN
			StateNext(work_data.state);
		END_IF
	201:
		IF cut_data.state = State.READY THEN
			supply_data.state_glue := State.RST;
			supply_data.state_conveyer := State.RST;
			supply_data.state_roll := State.RST;
			stick_data.state_roll := State.RST;
			cut_data.state := State.HOME;
			StateNext(work_data.state);
		END_IF
	202:
		IF (	supply_data.state_glue = State.READY AND
				supply_data.state_conveyer = State.READY AND
				supply_data.state_roll = State.READY AND
				stick_data.state_roll = State.RST_DONE AND
				cut_data.state = State.HOME_DONE
			) THEN
			stick_data.state_roll := State.HOME;
			StateNext(work_data.state);
		END_IF
	203:
		IF stick_data.state_roll = State.HOME_DONE THEN
			StateNext(work_data.state);
		END_IF
	204:
		IF work_data.halt.rise.Q THEN
			StateNext(work_data.state);
		END_IF
	205:
		supply_data.state_glue := State.RUN;
		supply_data.state_conveyer := State.RUN;
		supply_data.state_roll := State.RUN;
		stick_data.state_roll := State.READY;
		cut_data.state := State.READY;
		StateNext(work_data.state);
	206:
		IF (	supply_data.state_glue = State.RUN_ING AND
				supply_data.state_conveyer = State.RUN_ING AND
				supply_data.state_roll = State.RUN_ING
			) THEN
			work_data.state := State.RUN_ING;
		END_IF
END_CASE
END_ACTION

ACTION stick:
/////////
//PRESS//
/////////
CASE stick_data.state_press OF
	State.RST:
		stick_data.press.on := FALSE;
		StateNext(stick_data.state_press);
	2:
		IF stick_data.press.n_timer.Q THEN
			stick_data.state_press := State.READY;
		END_IF
	//////\\
	////\\\\
	//\\\\\\
	State.RUN:
		stick_data.press.on := TRUE;
		StateNext(stick_data.state_press);
	102:
		IF stick_data.press.p_timer.Q THEN
			stick_data.state_press := State.RUN_ING;
		END_IF
	//////\\
	////\\\\
	//\\\\\\
	State.RUN_ING:
		//
END_CASE

////////
//ROLL//
////////
CASE stick_data.state_roll OF
	State.RST:
		axis_stick_fv.bExecute := TRUE;
		axis_stick_mv.Velocity := axis_stick_fv.fSetVelocity;
		axis_stick_mv.Deceleration := stick_data.speed_target / c_axis_stick_ramp_time_sec;
		IF axis_stick_mv.Velocity > 0.0 THEN
			StateNext(stick_data.state_roll);
		ELSE
			stick_data.state_roll := 10;
		END_IF
	2:
		axis_stick_mv.Velocity := MAX(0.0, axis_stick_mv.Velocity - axis_stick_mv.Deceleration * c_dt);
		axis_stick_fv.fSetVelocity := axis_stick_mv.Velocity;
		IF axis_stick_mv.Velocity = 0.0 THEN
			stick_data.state_roll := 10;
		END_IF
	10:
		axis_stick_set_position.Position := 0.0;
		axis_stick_set_position.Execute := TRUE;
		StateNext(stick_data.state_roll);
	11:
		IF axis_stick_set_position.Done THEN
			axis_stick_set_position.Execute := FALSE;
			stick_data.state_roll := State.RST_DONE;
		END_IF
	//////\\
	////\\\\
	//\\\\\\
	State.HOME:
		stick_data.state_roll := State.HOME_DONE;
	//////\\
	////\\\\
	//\\\\\\
	State.READY:
		IF stick_data.foil_in_rise.Q THEN
			stick_data.state_roll := State.RUN;
		END_IF
	//////\\
	////\\\\
	//\\\\\\
	State.RUN:
		axis_stick_mv.Acceleration := stick_data.speed_target / c_axis_stick_ramp_time_sec;
		StateNext(stick_data.state_roll);
	102:
		axis_stick_mv.Velocity := MIN(axis_stick_mv.Velocity + axis_stick_mv.Acceleration * c_dt, stick_data.speed_target);
		axis_stick_fv.fSetVelocity := axis_stick_mv.Velocity * cut_data.speed_factor;
		IF stick_data.foil_in_fall.Q THEN
			stick_data.stop_distance := (
				(UDINT_TO_LREAL(save_data.stick_stop_distance_micron) * 1E3)
				/ stick_data.micron_per_servo_round
			);// + (stick_data.speed_target * c_axis_stick_ramp_time_sec * 0.5);
			axis_stick_mv.Deceleration := (
				(axis_stick_mv.Velocity * axis_stick_mv.Velocity)
				/ (2 * stick_data.stop_distance)
			);
			StateNext(stick_data.state_roll);
		END_IF
	103:
		axis_stick_mv.Velocity := MAX(0.0, axis_stick_mv.Velocity - axis_stick_mv.Deceleration * c_dt);
		axis_stick_fv.fSetVelocity := axis_stick_mv.Velocity * cut_data.speed_factor;
		IF axis_stick_mv.Velocity = 0.0 THEN
			StateNext(stick_data.state_roll);
		END_IF
	104:
		stick_data.state_roll := State.READY;
END_CASE
END_ACTION

END_PROGRAM

// Device/Application/StateNext
FUNCTION StateNext
VAR_INPUT
	state: REFERENCE TO INT;
END_VAR
VAR
END_VAR

state := state + 1;

END_FUNCTION

// Device/Application/Visualization
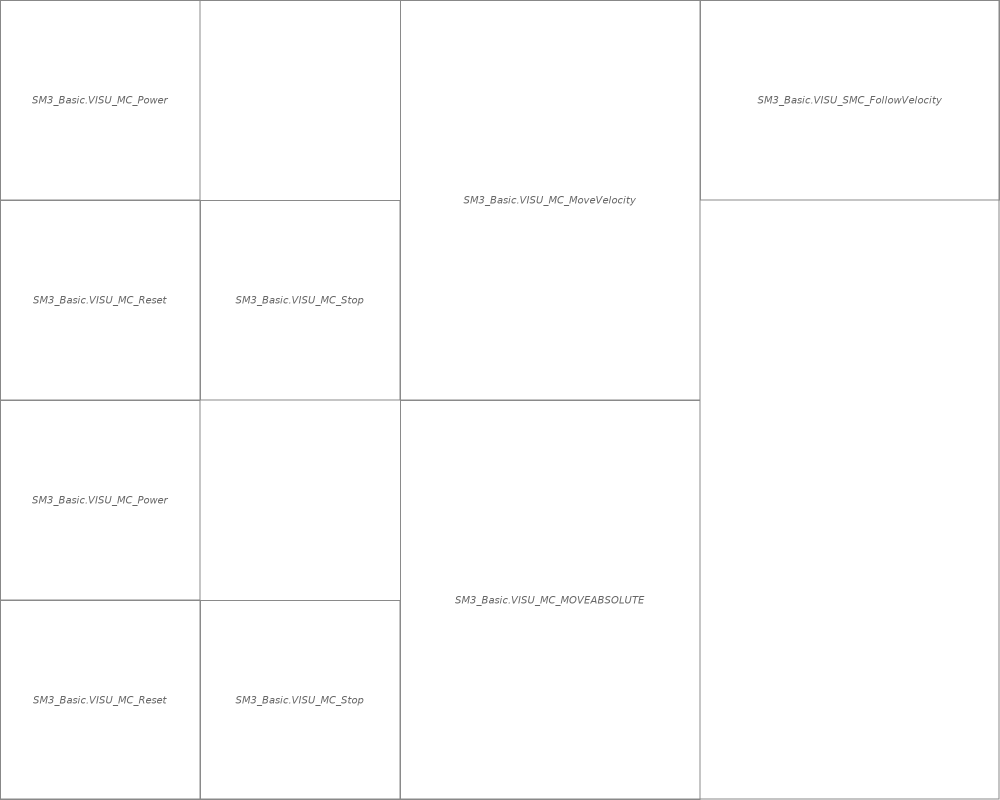
VISUALIZATION Visualization  // 1000x800
    Frame (0,0 200x200)
        shows SM3_Basic.VISU_MC_Power(m_Input_FB := main.axis_stick_power)
    Frame (0,200 200x200)
        shows SM3_Basic.VISU_MC_Reset(m_Input_FB := main.axis_stick_reset)
    Frame (200,200 200x200)
        shows SM3_Basic.VISU_MC_Stop(m_Input_FB := main.axis_stick_stop)
    Frame (400,400 300x400)
        shows SM3_Basic.VISU_MC_MOVEABSOLUTE(m_Input_FB := main.axis_cut_mabs)
    Frame (0,400 200x200)
        shows SM3_Basic.VISU_MC_Power(m_Input_FB := main.axis_cut_power)
    Frame (0,600 200x200)
        shows SM3_Basic.VISU_MC_Reset(m_Input_FB := main.axis_cut_reset)
    Frame (200,600 200x200)
        shows SM3_Basic.VISU_MC_Stop(m_Input_FB := main.axis_cut_stop)
    Frame (400,0 300x400)
        shows SM3_Basic.VISU_MC_MoveVelocity(m_Input_FB := main.axis_stick_mv)
    Frame (700,0 300x200)
        shows SM3_Basic.VISU_SMC_FollowVelocity(m_Input_FB := main.axis_stick_fv)
END_VISUALIZATION
